VAR_GLOBAL
	ads_watch_dog : FB_ADS_WATCHDOG;
END_VAR

(* stored: Version 1.1.0.1, ProductVersion 3.1.4024.2
   GVL GVL_VAC_INTF: Id {165b9a13-b466-4efc-8e82-d6aa491fa983} *)
